Staubli VAL3: OnF7.pgx

public program OnF7()
begin
end
